FUNCTION F_ITC_SendESR : BOOL
(**************************************************************************************
 * 	Application		:	BoxControl Framework
 *	Revision		:	$Revision: 404529 $
 *	Revision date	:	$Date: 2018-04-23 08:21:38 +0200 (Mo., 23 Apr 2018) $
 *	Last changed by	:	$Author: b7bolm $
 *	URL				:	$URL: http://almscdc.swisslog.com/repo/SWPD/Development/BoxControlFramework/20_Release/trunk/01_Software/BCF/BCF/JumpStart/20_Product/10_App/11_Com/10_Lib/10_Conv/11_ITC/F_ITC_SendESR.TcPOU $
 *
 *	Purpose			:	Wrap message - ESR
 *
 * ------------------------------------------------------------------------------------
 *	Copyright Swisslog [IP AG], Switzerland. All rights reserved.
 * 
 * ------------------------------------------------------------------------------------
 *	
 * 	Revision History: 
 *
 * 	VERSION			DATE			INITIALS			DESCRIPTION
 *	0.1				01.01.2001		swl					Example
 *
 **************************************************************************************)
VAR_INPUT
	eChannelSrc			: E_MFCS_Channel; // Source communicaton channel		
	ElementName	 		: STRING(Conveyor.POSITION_STRINGLENGTH); // SIS MM-GGG-EEEE-FF-Z
	eState				: E_PositionState; // State
	Enabled				: BOOL; // State
	eErrorState			: E_ErrorState; // Error State
	eErrorCode			: E_ErrorConv; // Return Code
	eErrorType			: E_ErrorType; // Error Type
	ErrorInformation	: STRING(System.ERROR_PARAM_STRINGLENGTH); // 5 Chars Error Information
	Variable			: DINT; // Variable
	eReturnCode			: E_ErrorConv; // Return code
END_VAR
VAR
	ESR					: ST_ITC_ESR; 
END_VAR

// Map values
ESR.Position := ElementName;
ESR.Enabled := Enabled;
ESR.State := eState;
ESR.Variable := Variable;
ESR.ErrorCode := eErrorCode;
ESR.ErrorInformation := ErrorInformation;
ESR.ErrorState := eErrorState;
ESR.ErrorType := eErrorType;
ESR.ReturnCode := eReturnCode;

// Forward to ITC
F_ITC_SendESR := fbITC_Manager.M_SendData(
					meChannel	:= eChannelSrc,
					mMsgType	:= E_ITC_MsgTypeConv.ELEMENT_STATUS_REPORT,
					mpData		:= ADR(ESR),
					mLen		:= SIZEOF(ESR));

END_FUNCTION

(* stored: Version 1.1.0.1, ProductVersion 3.1.4022.12
   POU F_ITC_SendESR: Id {e7801e4a-11a1-42f5-be8d-df32a16e73ae}, SpecialFunc None *)
